Fanuc KAREL source: kb00025.KL

-- PROVISIONAL review KL for V940-1; original PC SHA256 bfb1a033a84299ec9e892f0cb58e2c57fa9a08d75e21a4fadc9256c56e0a8057
-- Incomplete behavior may be omitted. Consult companion uncertainty JSON. Do not deploy.
PROGRAM KB00025
%NOLOCKGROUP
BEGIN
  -- V9_ZERO_TABLE_METADATA_HINT layout=0002_ascii; no indexed target words; source/name/runtime held
  -- UNRESOLVED_PC offsets 5-12; opcodes 9D,23
  -- UNRESOLVED_PC offsets 17-24; opcodes 9D,23
  -- UNRESOLVED_PC offsets 29-36; opcodes 9D,23
  -- UNRESOLVED_PC offsets 41-63; opcodes 27,22,22,22,31
  -- UNRESOLVED_PC offsets 68-72; opcodes 7F
END KB00025
